// TIA Portal project "modebus com" (V16)

(* hardware
DEVICE "S7-1200 station_1"  S7-1200 Station
   slot 0: "Rack_0"  S7-1200 Rack  Rack  V1.0
   slot 1: "PLC_1"  CPU 1211C DC/DC/DC  6ES7 211-1AE40-0XB0  V4.4
   slot 3: "CB 1241 (RS485)"  CB 1241 (RS485)  6ES7 241-1CH30-1XB0  V1.0
*)

// ===== PLC "PLC_1"  CPU 1211C DC/DC/DC =====

VAR_GLOBAL   // PLC tag table "Default tag table"
   "System_Byte" AT %MB0 : Byte;
   "FirstScan" AT %M0.0 : Bool;
   "DiagStatusUpdate" AT %M0.1 : Bool;
   "AlwaysTRUE" AT %M0.2 : Bool;
   "AlwaysFALSE" AT %M0.3 : Bool;
   "Clock_Byte" AT %MB1 : Byte;
   "Clock_10Hz" AT %M1.0 : Bool;
   "Clock_5Hz" AT %M1.1 : Bool;
   "Clock_2.5Hz" AT %M1.2 : Bool;
   "Clock_2Hz" AT %M1.3 : Bool;
   "Clock_1.25Hz" AT %M1.4 : Bool;
   "Clock_1Hz" AT %M1.5 : Bool;
   "Clock_0.625Hz" AT %M1.6 : Bool;
   "Clock_0.5Hz" AT %M1.7 : Bool;
   "Tag_1" AT %M20.0 : Bool;
   "Tag_2" AT %MW100 : Int;
   "Control_Word" AT %MW10 : Word;
   "Speed_Value" AT %MW12 : Word;
   "Output_Freqyency" AT %MW14 : Word;
   "Output_ Current" AT %MW16 : Word;
   "Run_Forward" AT %M2.0 : Bool;
   "Run_Reverse" AT %M2.1 : Bool;
   "Stop" AT %M2.2 : Bool;
   "Reset_Fault" AT %M2.3 : Bool;
   "Hmi_Frequency" AT %MD60 : Real;
   "Tag_4" AT %MD64 : Real;
   "Tag_3" AT %MD68 : Real;
   "frequency_valueHMI" AT %MD72 : Real;
   "Tag_5" AT %MD74 : Real;
   "Current_ValueHMI" AT %MD78 : Real;
END_VAR

// folder: System blocks/Program resources

DATA_BLOCK "IEC_Counter_0_DB"   // DB2
{ S7_Optimized_Access := 'TRUE' }
AUTHOR : Simatic
FAMILY : IEC
NAME : CNTR
VERSION : 1.0
// stored: InstanceOfName IEC_COUNTER
"IEC_COUNTER"
BEGIN
END_DATA_BLOCK

// folder: (top level)

ORGANIZATION_BLOCK "Main"   // OB1, LAD, ProgramCycle
TITLE = "Main Program Sweep (Cycle)"
{ S7_Optimized_Access := 'TRUE' }
VERSION : 0.1
   VAR_INPUT
      Initial_Call : Bool;   // Initial call of this OB
      Remanence : Bool;   // =True, if remanent data are available
   END_VAR
BEGIN

REGION Network 1: connection counter
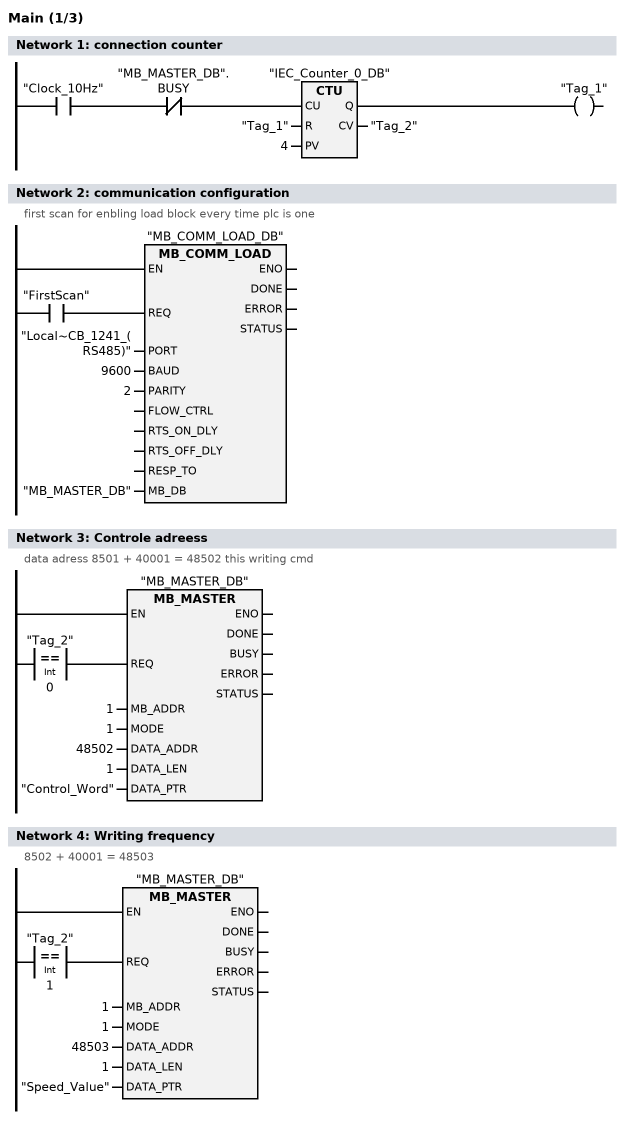
   "IEC_Counter_0_DB".CTU(CU := "Clock_10Hz" AND NOT "MB_MASTER_DB".BUSY, R := "Tag_1", PV := 4, CV => "Tag_2");
   "Tag_1" := "IEC_Counter_0_DB".Q;
END_REGION

REGION Network 2: communication configuration
   // first scan for enbling load block every time plc is one
   "MB_COMM_LOAD_DB"(REQ := "FirstScan",   // MB_COMM_LOAD
                     PORT := "Local~CB_1241_(RS485)",
                     BAUD := 9600,
                     PARITY := 2,
                     MB_DB := "MB_MASTER_DB");
END_REGION

REGION Network 3: Controle adreess
   // data adress 8501 + 40001 = 48502 this writing cmd
   "MB_MASTER_DB"(REQ := "Tag_2" = 0,   // MB_MASTER
                  MB_ADDR := 1,
                  MODE := 1,
                  DATA_ADDR := 48502,
                  DATA_LEN := 1,
                  DATA_PTR := "Control_Word");
END_REGION

REGION Network 4: Writing frequency
   // 8502 + 40001 = 48503
   "MB_MASTER_DB"(REQ := "Tag_2" = 1,   // MB_MASTER
                  MB_ADDR := 1,
                  MODE := 1,
                  DATA_ADDR := 48503,
                  DATA_LEN := 1,
                  DATA_PTR := "Speed_Value");
END_REGION

REGION Network 5: reading output frequency so mode = 0
   // 4000 + 3202 = 43203
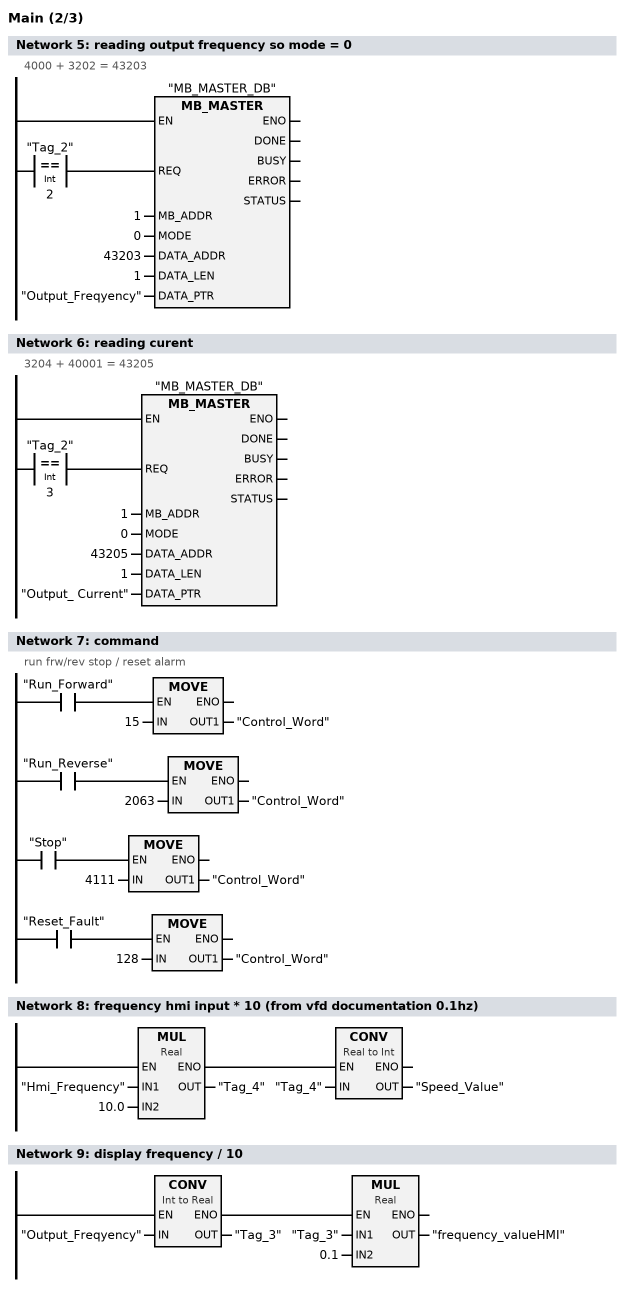
   "MB_MASTER_DB"(REQ := "Tag_2" = 2,   // MB_MASTER
                  MB_ADDR := 1,
                  MODE := 0,
                  DATA_ADDR := 43203,
                  DATA_LEN := 1,
                  DATA_PTR := "Output_Freqyency");
END_REGION

REGION Network 6: reading curent
   // 3204 + 40001 = 43205
   "MB_MASTER_DB"(REQ := "Tag_2" = 3,   // MB_MASTER
                  MB_ADDR := 1,
                  MODE := 0,
                  DATA_ADDR := 43205,
                  DATA_LEN := 1,
                  DATA_PTR := "Output_ Current");
END_REGION

REGION Network 7: command
   // run frw/rev stop / reset alarm
   RUNG wire#powerrail
      Contact( "Run_Forward" )
      Move(in := 15, out1 => "Control_Word")
   END_RUNG
   RUNG wire#powerrail
      Contact( "Run_Reverse" )
      Move(in := 2063, out1 => "Control_Word")
   END_RUNG
   RUNG wire#powerrail
      Contact( "Stop" )
      Move(in := 4111, out1 => "Control_Word")
   END_RUNG
   RUNG wire#powerrail
      Contact( "Reset_Fault" )
      Move(in := 128, out1 => "Control_Word")
   END_RUNG
   // the same network as SCL:
   IF "Run_Forward" THEN "Control_Word" := 15; END_IF;
   IF "Run_Reverse" THEN "Control_Word" := 2063; END_IF;
   IF "Stop" THEN "Control_Word" := 4111; END_IF;
   IF "Reset_Fault" THEN "Control_Word" := 128; END_IF;
END_REGION

REGION Network 8: frequency hmi input * 10 (from vfd documentation 0.1hz)
   RUNG wire#powerrail
      { S7_Templates := "SrcType := Real" } Mul(in1 := "Hmi_Frequency", in2 := 10.0, out => "Tag_4")
      { S7_Templates := "[SrcType := Real, DestType := Int]" } Convert(in := "Tag_4", out => "Speed_Value")
   END_RUNG
   // the same network as SCL:
   "Tag_4" := "Hmi_Frequency" * 10.0;
   "Speed_Value" := REAL_TO_INT("Tag_4");
END_REGION

REGION Network 9: display frequency / 10
   RUNG wire#powerrail
      { S7_Templates := "[SrcType := Int, DestType := Real]" } Convert(in := "Output_Freqyency", out => "Tag_3")
      { S7_Templates := "SrcType := Real" } Mul(in1 := "Tag_3", in2 := 0.1, out => "frequency_valueHMI")
   END_RUNG
   // the same network as SCL:
   "Tag_3" := INT_TO_REAL("Output_Freqyency");
   "frequency_valueHMI" := "Tag_3" * 0.1;
END_REGION

REGION Network 10: display current on hmi
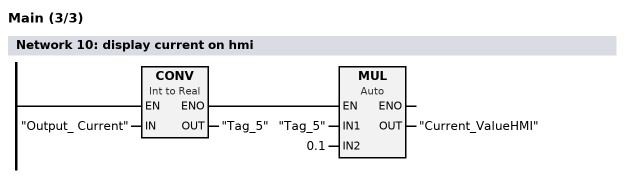
   RUNG wire#powerrail
      { S7_Templates := "[SrcType := Int, DestType := Real]" } Convert(in := "Output_ Current", out => "Tag_5")
      Mul(in1 := "Tag_5", in2 := 0.1, out => "Current_ValueHMI")
   END_RUNG
   // the same network as SCL:
   "Tag_5" := INT_TO_REAL("Output_ Current");
   "Current_ValueHMI" := "Tag_5" * 0.1;
END_REGION
END_ORGANIZATION_BLOCK